// TIA Portal V17 export
// export: Created 2025-06-26T07:49:49.032974Z, ExportSetting WithDefaults, DisplayName Totally Integrated Automation Portal, DisplayVersion V17 Update 8, DisplayName TIA Portal Openness, DisplayVersion V17 Update 8, DisplayName TIA Portal Version Control Interface, DisplayVersion V17, DisplayName STEP 7 Professional, DisplayVersion V17 Update 8, DisplayName STEP 7 Safety, DisplayVersion V17 Update 6, DisplayName WinCC Advanced, DisplayVersion V17 Update 8
FUNCTION_BLOCK "fbDeviationAlarm"   // FB55, FBD
{ S7_Optimized_Access := 'TRUE' }
AUTHOR : Heaten
VERSION : 0.1
// stored: AutoNumber true, IsIECCheckEnabled false, IsRetainMemResEnabled false, MemoryReserve 0, SetENOAutomatically false, UDAEnableTagReadback false
   VAR_INPUT
      sActualValue : "stCalcValue";   // Process value
      fCommandValue : Real;   // Setpoint
      bAckAll : Bool;
      bEnable : Bool;
   END_VAR
   VAR_IN_OUT
      sTag : "stDeviationAlarm";
   END_VAR
   VAR
      Alarm : "fbAlarm";
   END_VAR
   VAR_TEMP
      AlarmCondition : Bool;
   END_VAR
BEGIN

REGION Network 1 (SCL): Alarm condition if measured value ok
   IF #sActualValue.bError = FALSE THEN
       #AlarmCondition := ABS(#sActualValue.fValue - #fCommandValue) > #sTag.fDeviationLimit;
   ELSE
       #AlarmCondition := FALSE;
   END_IF;
END_REGION

REGION Network 2: Alarm with activation delay
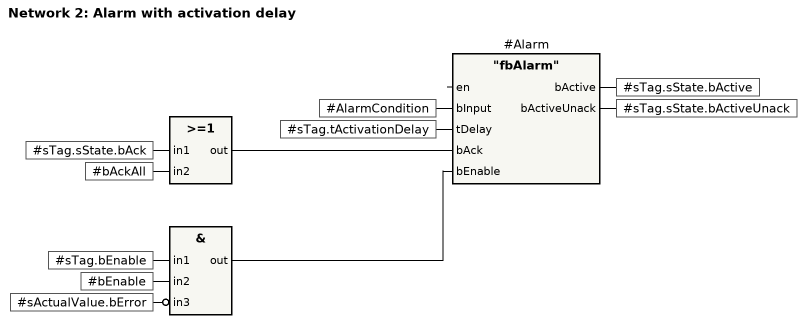
   #Alarm(bInput := #AlarmCondition,   // "fbAlarm"
          tDelay := #sTag.tActivationDelay,
          bAck := #sTag.sState.bAck OR #bAckAll,
          bEnable := #sTag.bEnable AND #bEnable AND NOT #sActualValue.bError,
          bActive => #sTag.sState.bActive,
          bActiveUnack => #sTag.sState.bActiveUnack);
END_REGION
END_FUNCTION_BLOCK
